FUNCTION_BLOCK FB_ModbusRtuMaster_KL6x22B //IMPLEMENTS I_UniversalUnit
VAR
	sName			:		STRING;
	iScantime		:		UINT := 50;
	iTimeout		:		UINT := 1000;//1000ms
	iErrorID		:		MODBUS_ERRORS;
	bBusy			: 		BOOL;
	bError			:		BOOL;
	iStepGeneral	: 		E_ModBusMasterState;
	iStepRunning	:		E_ModbusMasterStateRun;
	bFirstCycle		:		BOOL;
	bStop			: 		BOOL;

	fbModbusMaster	: 		ModbusRtuMaster_KL6x22B;
	ipModbusSlave	:		ARRAY [1..247] OF I_ModbusSlaveRtu;
	iAmountSlave	: 		UINT;
	
	iLoopSlave		:		UINT	:= 1;
	iLoopAdr		:		UINT;
	iQuantity 		: 		POINTER TO WORD;
	iMBAddr 		: 		POINTER TO WORD;
    arrData			: 		ARRAY [0..255] OF WORD;
	
	UnitId			: BYTE;
	Quantity		: WORD;
	MBAddr			: WORD;
	cbLength 		: UINT;
	pMemoryAddr		: POINTER TO BYTE;
	pDataWrite		: POINTER TO WORD;

	bexecute		: BOOL;
	
	tCalculateTimeRW	: TON;
	tTimerScanDelay		: TON;
	nNumberFaultRW		: UINT;
	eModbusFunction		: E_ModbusFunction;
	peModbusFunction 	: POINTER TO WORD;
END_VAR

StateMachine();
iErrorID := fbModbusMaster.ErrorId;

PROPERTY AnyError : BOOL
GET
AnyError 	:= bError;
END_GET
END_PROPERTY

PROPERTY Busy : BOOL
GET
Busy := bBusy;
END_GET
END_PROPERTY

PROPERTY CycleTimeMeasure : Time
GET
CycleTimeMeasure := tCalculateTimeRW.ET;
END_GET
END_PROPERTY

PROPERTY ErrorID : MODBUS_ERRORS
GET
ErrorID := iErrorID;
END_GET
END_PROPERTY

PROPERTY Name : STRING
GET
Name := sName;
END_GET
SET
sName := Name;
END_SET
END_PROPERTY

PROPERTY ReadData : ARRAY [0..255] OF Word
GET
ReadData := arrData;
END_GET
END_PROPERTY

PROPERTY ReadDataSize : uint
GET
ReadDataSize := INT_TO_UINT(SIZEOF(arrData));
END_GET
END_PROPERTY

METHOD RegisterSlave : BOOL
VAR_INPUT
	ModbusSlave		:		I_ModbusSlaveRtu;
END_VAR
VAR
	iLoop	:	UINT;
	bExists	:	BOOL;
END_VAR
FOR iLoop := 1 TO iAmountSlave DO
	IF ipModbusSlave[iLoop] = ModbusSlave THEN
		bExists := TRUE;
		iLoop := iAmountSlave;// end loop for command
	END_IF
END_FOR 
IF NOT bExists THEN
	iAmountSlave := iAmountSlave + 1;
	ipModbusSlave[iAmountSlave] := ModbusSlave;
END_IF
END_METHOD

METHOD Reset : BOOL
bError := FALSE;
iErrorID := 0;
bError := FALSE;
iStepGeneral := E_ModBusMasterState.Stop;
iStepRunning := E_ModbusMasterStateRun.CheckNumberSlaveRegistered;
iLoopSlave := 1;
iLoopAdr := 0;
fbModbusMaster.Execute := FALSE;
Reset := TRUE;
END_METHOD

METHOD Run : BOOL /// call from FB_modbus
iStepGeneral := E_ModBusMasterState.Running;
Run := TRUE;
END_METHOD

PROPERTY ScanTime : UINT
GET
ScanTime := iScantime;
END_GET
SET
iScantime := ScanTime;
END_SET
END_PROPERTY

METHOD protected StateMachine : BOOL (*State machine of unit*)
CASE iStepGeneral OF
	E_ModBusMasterState.stop:
		StateStopping();
			
	E_ModBusMasterState.Running: 
		StateRunning();
END_CASE
END_METHOD

METHOD PROTECTED StateRunning : BOOL (* Unit is uninitialized*)
VAR 
	

	
END_VAR
CASE iStepRunning OF
	E_ModbusMasterStateRun.CheckNumberSlaveRegistered: // Trigger
		tCalculateTimeRW(
			IN := TRUE,
			PT := T#5M
		);	
		IF iAmountSlave > 0 THEN
			iStepRunning := E_ModbusMasterStateRun.SetParametersRead;
		END_IF
			
	E_ModbusMasterStateRun.SetParametersRead: // Set parameters
		IF ipModbusSlave[iLoopSlave].NumAddRegionRead <> 0 
		AND iLoopAdr <= (ipModbusSlave[iLoopSlave].NumAddRegionRead - 1) 
		THEN
			iQuantity := ipModbusSlave[iLoopSlave].AddressRead + ((iLoopAdr * 3 + 1) * SIZEOF(WORD));// arrAddressRead[iloopAdr][1] in Slave
			iMBAddr := ipModbusSlave[iLoopSlave].AddressRead + ((iLoopAdr * 3) * SIZEOF(WORD));// arrAddressRead[iloopAdr][0] in Slave
			UnitID := ipModbusSlave[iLoopSlave].UnitID;
			Quantity :=	iQuantity^;
			MBAddr := iMBAddr^;
			cbLength := SIZEOF(arrData);
			pMemoryAddr	:= ADR(arrData);
			peModbusFunction := ipModbusSlave[iLoopSlave].AddressRead + ((iLoopAdr * 3 + 2) * SIZEOF(WORD)); // arrAddressRead[iloopAdr][2] in Slave
			eModbusFunction := peModbusFunction^;
			iStepRunning := E_ModbusMasterStateRun.SendRequestRead;
		ELSE 
			iLoopAdr := 0;
			iStepRunning := E_ModbusMasterStateRun.ReturnReadDone;
		END_IF

			
	E_ModbusMasterStateRun.SendRequestRead: // Send request
		CASE eModbusFunction OF
			E_ModbusFunction.ReadHoldingRegisters:
				fbModbusMaster.ReadRegs(
					UnitID:= UnitID, 
					Quantity:= Quantity, 
					MBAddr:= MBAddr, 
					cbLength:= cbLength, 
					pMemoryAddr:= pMemoryAddr, 
					Execute:= TRUE,
					Timeout:= UINT_TO_TIME(iTimeout),
					BUSY=> bBusy, 
					Error=> bError , 
					ErrorId=>iErrorId 
				);
			
			E_ModbusFunction.ReadInputRegisters:
				fbModbusMaster.ReadInputRegs(
					UnitID:= UnitID, 
					Quantity:= Quantity, 
					MBAddr:= MBAddr, 
					cbLength:= cbLength, 
					pMemoryAddr:= pMemoryAddr, 
					Execute:= TRUE,
					Timeout:= UINT_TO_TIME(iTimeout),
					BUSY=> bBusy, 
					Error=> bError , 
					ErrorId=>iErrorId 
				);
			
		END_CASE
		iStepRunning := E_ModbusMasterStateRun.WaitReadRespond;
						
	E_ModbusMasterStateRun.WaitReadRespond:
		fbModbusMaster.ReadRegs(Execute := FALSE);
		fbModbusMaster.ReadInputRegs(Execute := FALSE);
		IF NOT fbModbusMaster.BUSY AND NOT fbModbusMaster.Error THEN
			ipModbusSlave[iLoopSlave].ModbusErrorID := iErrorID;
			iStepRunning := E_ModbusMasterStateRun.ConvertRawData;
			nNumberFaultRW := 0;
		END_IF
		
		IF fbModbusMaster.Error AND NOT fbModbusMaster.BUSY THEN
			ipModbusSlave[iLoopSlave].ModbusErrorID := iErrorID;
			iStepRunning := E_ModbusMasterStateRun.ReturnReadDone;
		END_IF
	
	E_ModbusMasterStateRun.ConvertRawData: 
		ipModbusSlave[iLoopSlave].Convert(
			iRegionNo := iLoopAdr,
		 	pReadData := ADR(arrData)
		);
		iLoopAdr := iLoopAdr + 1;
		iStepRunning := E_ModbusMasterStateRun.CheckNumberSlaveRegistered;

	E_ModbusMasterStateRun.ReturnReadDone: // Return, done
		iStepRunning := E_ModbusMasterStateRun.SetParametersWrite;
		iLoopAdr := 0;

	E_ModbusMasterStateRun.SetParametersWrite :
		IF  ipModbusSlave[iLoopSlave].NumAddRegionWrite <> 0
		AND iLoopAdr <= ipModbusSlave[iLoopSlave].NumAddRegionWrite - 1 
		THEN // iLoopAdr start from 1
			iMBAddr := ipModbusSlave[iLoopSlave].AddressWrite + (iLoopAdr * 11 * SIZEOF(WORD));// return address word contain value address( modbus) 
			pDataWrite := ipModbusSlave[iLoopSlave].AddressWrite + ((iLoopAdr * 11 + 2) * SIZEOF(WORD));
			iQuantity := ipModbusSlave[iLoopSlave].AddressWrite + ((iLoopAdr * 11 + 1) * SIZEOF(WORD));
			peModbusFunction := ipModbusSlave[iLoopSlave].AddressWrite + ((iLoopAdr * 11 + 10) * SIZEOF(WORD));
			eModbusFunction := peModbusFunction^;
			UnitID 	:=		ipModbusSlave[iLoopSlave].UnitID;
			Quantity	:=	iQuantity^;
			MBAddr	:=		iMBAddr^;
			cbLength	:= 	Quantity * 2;
			pMemoryAddr	:= 	pDataWrite;
			iStepRunning := E_ModbusMasterStateRun.SendRequestWrite;
		ELSE 
			iStepRunning := E_ModbusMasterStateRun.ReturnWriteDone;
		END_IF

	E_ModbusMasterStateRun.SendRequestWrite :
		CASE eModbusFunction OF
			E_ModbusFunction.WriteMultipleCoils:
				fbModbusMaster.WriteMultipleCoils(
					UnitID:= UnitID, 
					Quantity:= Quantity, 
					MBAddr:= MBAddr, 
					cbLength:= cbLength, 
					pMemoryAddr:= pMemoryAddr, 
					Execute:=  true,
					Timeout:= 	UINT_TO_TIME(iTimeout),	
					BUSY=> bBusy, 
					Error=> bError , 
					ErrorId=>iErrorId 
				);
													
			E_ModbusFunction.WriteMultipleRegisters:
				fbModbusMaster.WriteRegs(
					UnitID:= UnitID, 
					Quantity:= Quantity, 
					MBAddr:= MBAddr, 
					cbLength:= cbLength, 
					pMemoryAddr:= pMemoryAddr, 
					Execute:= TRUE,
					Timeout:= UINT_TO_TIME(iTimeout),	
					BUSY=> bBusy, 
					Error=> bError , 
					ErrorId=>iErrorId 
				);
											
			E_ModbusFunction.WriteSingleCoil:
				fbModbusMaster.WriteSingleCoil(
					UnitID:= UnitID, 
					Quantity:= Quantity, 
					MBAddr:= MBAddr, 
					cbLength:= cbLength, 
					pMemoryAddr:= pMemoryAddr, 
					Execute:=  true,
					Timeout:= UINT_TO_TIME(iTimeout),	
					BUSY=> bBusy, 
					Error=> bError , 
					ErrorId=>iErrorId 
				);
			E_ModbusFunction.WriteSingleRegister:
				fbModbusMaster.WriteSingleRegister(
					UnitID:= UnitID, 
					Quantity:= Quantity, 
					MBAddr:= MBAddr, 
					cbLength:= cbLength, 
					pMemoryAddr:= pMemoryAddr, 
					Execute:=  true,
					Timeout:= 	UINT_TO_TIME(iTimeout),	
					BUSY=> bBusy, 
					Error=> bError , 
					ErrorId=>iErrorId 
				);
		END_CASE
		
		iStepRunning := E_ModbusMasterStateRun.WaitWriteRespond;
	
	E_ModbusMasterStateRun.WaitWriteRespond :
		fbModbusMaster.WriteMultipleCoils( Execute := FALSE);
		fbModbusMaster.WriteRegs( Execute := FALSE);
		fbModbusMaster.WriteSingleCoil( Execute := FALSE);	
		fbModbusMaster.WriteSingleRegister( Execute := FALSE);
		IF NOT fbModbusMaster.BUSY AND NOT fbModbusMaster.Error THEN
			ipModbusSlave[iLoopSlave].ModbusErrorID := iErrorID;
			iStepRunning := E_ModbusMasterStateRun.SetParametersWrite;
			nNumberFaultRW := 0;
			iLoopAdr := iLoopAdr + 1;
		END_IF
		IF fbModbusMaster.Error AND NOT fbModbusMaster.BUSY THEN
			ipModbusSlave[iLoopSlave].ModbusErrorID := iErrorID;
			iStepRunning := E_ModbusMasterStateRun.ReturnWriteDone ;
		END_IF
	
	 E_ModbusMasterStateRun.ReturnWriteDone :
		iLoopAdr := 0;
		iLoopSlave := iLoopSlave + 1;// next slave
		IF iLoopSlave > iAmountSlave THEN
			iLoopSlave := 1;
		END_IF
		tTimerScanDelay( 
			IN := TRUE,
			PT := UINT_TO_TIME(iScantime)
		);
		IF tTimerScanDelay.Q THEN
			tTimerScanDelay( IN := FALSE);
			tCalculateTimeRW(in := FALSE);
		 	iStepRunning := E_ModbusMasterStateRun.CheckNumberSlaveRegistered;
		END_IF
			
END_CASE
END_METHOD

METHOD protected StateStopping : BOOL (* Unit is uninitialized*)
iStepRunning	:= E_ModbusMasterStateRun.CheckNumberSlaveRegistered;
iLoopSlave		:= 1;
iLoopAdr		:= 0;
fbModbusMaster.WriteMultipleCoils( Execute := FALSE);
fbModbusMaster.WriteRegs( Execute := FALSE);
fbModbusMaster.WriteSingleCoil( Execute := FALSE);	
fbModbusMaster.WriteSingleRegister( Execute := FALSE);
fbModbusMaster.ReadRegs(Execute := FALSE);
fbModbusMaster.ReadInputRegs(Execute := FALSE);
END_METHOD

METHOD Stop : BOOL
iStepGeneral := E_ModBusMasterState.stop;
Stop := TRUE;
END_METHOD

PROPERTY Stopped : bool
GET
Stopped := bStop;
END_GET
END_PROPERTY

PROPERTY Timeout : UINT // in milisecond, if not respond in this time , error will raise
GET
Timeout := iTimeout;
END_GET
SET
iTimeout := Timeout;
END_SET
END_PROPERTY

END_FUNCTION_BLOCK

(* stored: Version 1.1.0.1, ProductVersion 3.1.4024.12
   POU FB_ModbusRtuMaster_KL6x22B: Id {8e753c28-1fce-4d27-b11f-e9a15231152b}, SpecialFunc None
   Folder Methods: Id {47a6095f-578e-4588-a897-55e800c9935c}
   Folder Property: Id {d7edfaf2-f1c6-4e1e-b0ae-6f79dcd777e5}
   Folder StateMachine: Id {fedae15b-fa36-43f6-acdd-7488c867bb01}
   Property AnyError: Id {28006fca-c385-4865-8046-179a879c2c41}
   Get Get: Id {86b2de52-1cf0-40a4-b962-61621fc185fd}
   Property Busy: Id {4e627418-7181-4d2c-9d1a-3c8f4c4dfb08}
   Get Get: Id {5524bde0-2db7-4689-b5f7-3ec68ed53fc7}
   Property CycleTimeMeasure: Id {92667ac3-036d-4905-8d49-969c27da338b}
   Get Get: Id {1a5a3291-01d7-41ad-86b1-ce9c46c6fd76}
   Property ErrorID: Id {b775527a-6798-476d-bfa6-2c8081126d79}
   Get Get: Id {24c652ec-1402-4238-903c-1557c1ca5377}
   Property Name: Id {3d6a1954-4799-4748-b4d4-9987b1d4df00}
   Get Get: Id {76de1f64-2c0b-4e1a-8e9a-11cc296e1356}
   Set Set: Id {abb2c678-0126-49e5-8e87-47ab439a07cc}
   Property ReadData: Id {e47b5135-2aa3-40ec-a1de-a6b6f2e8df78}
   Get Get: Id {8d9cf0e9-db40-4487-870f-e10ed459e638}
   Property ReadDataSize: Id {e132369f-1805-4891-8836-346efcb36230}
   Get Get: Id {a0b858dc-4da5-48dc-add3-33946322a5a3}
   Method RegisterSlave: Id {2e0e4c13-ff3c-40bb-91b3-210a49a798b2}
   Method Reset: Id {816b3c00-ee72-4f2a-aab1-5ea67a249619}
   Method Run: Id {2a20e21f-52db-4d25-b2a3-fe58e91eb89c}
   Property ScanTime: Id {89f08984-48f4-4407-acfb-86c15773baef}
   Get Get: Id {158173c8-e928-4aac-8d83-7c1efa564534}
   Set Set: Id {ca95a500-53a5-4a5b-aff6-47701f7afb9e}
   Method StateMachine: Id {b3b7b051-4208-4c49-ad72-221b2c180cec}
   Method StateRunning: Id {de2556f8-a3a7-4507-8331-d1fee97b6a32}
   Method StateStopping: Id {5e0ec1ba-97e2-4383-a818-c21ad6a32e71}
   Method Stop: Id {9a90db34-d61c-425d-8c6f-be596019cd76}
   Property Stopped: Id {ee9dd436-ab02-4f7a-a904-f153256059a6}
   Get Get: Id {04198d20-306d-43e9-acc0-479aa7d3d09a}
   Property Timeout: Id {8eec85b2-20b9-4e88-aa4c-5d97157bbd3f}
   Get Get: Id {a0636adf-7e51-4faa-bd29-e19fc05b3c44}
   Set Set: Id {1be3caef-94ce-4479-933a-1a3f928ab18c} *)
